// TIA Portal V19 export
FUNCTION_BLOCK "TYPIC_C402_IF_M33"   // FB110, FBD
TITLE = TYPIC_C402_IF_M33: Voorwaarschuwingsbord
{ S7_Optimized_Access := 'TRUE' }
AUTHOR : OCOTECH
FAMILY : Typical
NAME : C402.703
// Logisch Object Besturing: C402.703
// 
// De interne functie M33 verzorgt de interne besturing van een M33obord.
// 
// Een M33obord is een waarschuwingsbord “verkeerslichten”. Dit bord waarschuwt het verkeer dat zij een actief verkeerslicht naderen.
// 
// Via het DVMosysteem worden de storingsmeldingen van ieder M33obord ingelezen. DVM meldt op zijn beurt storingen van iedere M33obord rechtstreeks aan 3B. De interne besturing heeft geen communicatie met DVM.
// stored: MemoryReserve 10, SetENOAutomatically false
   VAR_INPUT
      EXT_AUT { ExternalAccessible := 'False'; ExternalVisible := 'False'; ExternalWritable := 'False'} : Bool;   // Externe (hoofd) beveiliging (1 = OK)
      EXT_HW { ExternalAccessible := 'False'; ExternalVisible := 'False'; ExternalWritable := 'False'} : Bool;   // Sturings hardware (PLC) bewaking (1 = OK)
      IN_STO_NOK { ExternalAccessible := 'False'; ExternalVisible := 'False'; ExternalWritable := 'False'} : Bool;   // Storing aanwezig die niet observeerbaar tot gevolg heeft
      IN_STO_OK { ExternalAccessible := 'False'; ExternalVisible := 'False'; ExternalWritable := 'False'} : Bool;   // Storing aanwezig die observeerbaarheid niet beinvloed
      IN_PRTG_STO { ExternalAccessible := 'False'; ExternalVisible := 'False'; ExternalWritable := 'False'} : Bool;   // Storingsmelding RSS-bord vanuit PRTG
      IN_AUT_C402 { ExternalAccessible := 'False'; ExternalVisible := 'False'; ExternalWritable := 'False'} : Bool;   // Serie geschakelde beveiligingen (1 = OK)
      IN_AAN { ExternalAccessible := 'False'; ExternalVisible := 'False'; ExternalWritable := 'False'} : Bool;   // Terugmelding aansturing M33-bord (1 = AAN)
      CFG_TYD_FB { ExternalAccessible := 'False'; ExternalVisible := 'False'; ExternalWritable := 'False'} : Time;   // Vertragingstijd storing foute terugmelding
   END_VAR
   VAR_OUTPUT
      VAR_IF_M33 { ExternalAccessible := 'False'; ExternalVisible := 'False'; ExternalWritable := 'False'} : "C402_VAR_IF_M33_TYPIC";   // Struct met alle variabelen naar bovenliggende functies
      OUT_AAN { ExternalAccessible := 'False'; ExternalVisible := 'False'; ExternalWritable := 'False'} : Bool;   // Aansturing M33-bord (TRUE = Uit / FALSE = Aan)
   END_VAR
   VAR_IN_OUT
      STU_IF_M33 : "C402_STU_IF_M33_TYPIC";   // Struct met alle sturingen van de subfunctie (SF) M33 van 3B
   END_VAR
   VAR
      STO { ExternalWritable := 'False'} : Struct   // Storingen
         A001 { ExternalAccessible := 'False'; ExternalVisible := 'False'} : Bool;   // Beveiliging aangesproken
         A002 { ExternalAccessible := 'False'; ExternalVisible := 'False'} : Bool;   // Storing M33-bord gedetecteerd door PRTG
         A003 { ExternalAccessible := 'False'; ExternalVisible := 'False'} : Bool;   // Storing M33-bord
         A004 { ExternalAccessible := 'False'; ExternalVisible := 'False'} : Bool;   // Algemene storing M33-bord
         AT01 { ExternalAccessible := 'False'; ExternalVisible := 'False'} : Bool;   // Foute terugmelding: M33-bord aangestuurd, terugmelding Aan niet (of te laat) ontvangen
         AT02 { ExternalAccessible := 'False'; ExternalVisible := 'False'} : Bool;   // Foute terugmelding: M33-bord niet aangestuurd, terugmelding Aan blijft aanwezig
      END_STRUCT;
      VAR { ExternalWritable := 'False'} : Struct   // Variabelen
         STS_AAN { ExternalAccessible := 'False'; ExternalVisible := 'False'} : Bool;   // TRUE = M33-bord actueel in werking FALSE = Uit
         EXT_AUT { ExternalAccessible := 'False'; ExternalVisible := 'False'} : Bool;   // Externe (hoofd) beveiliging aangesproken
         EXT_HW { ExternalAccessible := 'False'; ExternalVisible := 'False'} : Bool;   // Sturings hardware (PLC) in storing
      END_STRUCT;
   END_VAR
BEGIN

REGION Network 1: START
END_REGION

REGION Network 2: +++ Aansturing bord +++
   // Aansturen bord en terugmeldingsbewaking (Aan / Uit).
END_REGION

REGION Network 3: +++ Storingen +++
   // Verwerken van de storingsmeldingen.
END_REGION

REGION Network 4: Storing A001: Beveiliging aangesproken
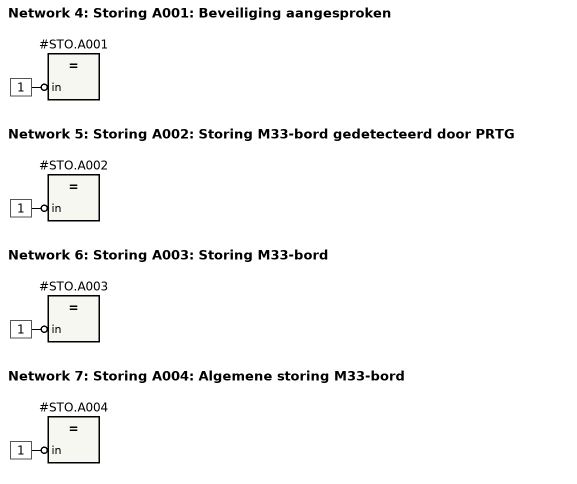
   #STO.A001 := NOT 1;
END_REGION

REGION Network 5: Storing A002: Storing M33-bord gedetecteerd door PRTG
   #STO.A002 := NOT 1;
END_REGION

REGION Network 6: Storing A003: Storing M33-bord
   #STO.A003 := NOT 1;
END_REGION

REGION Network 7: Storing A004: Algemene storing M33-bord
   #STO.A004 := NOT 1;
END_REGION

REGION Network 8 (SCL): EINDE
   // Variabelen van intern scada rakvlak naar outputs copieren
   #VAR_IF_M33.STS_AAN := #VAR.STS_AAN;
   #VAR_IF_M33.EXT_AUT := #VAR.EXT_AUT;
   #VAR_IF_M33.EXT_HW := #VAR.EXT_HW;
   #VAR_IF_M33.STO := #STO;
END_REGION
END_FUNCTION_BLOCK
